PROGRAM PRG_PLC2
VAR
	EncoderValue AT %I* : UINT;
	Pos					: LREAL;
END_VAR

F_ConsumeTime(20);

Pos:= UINT_TO_LREAL(EncoderValue)*100;

END_PROGRAM

(* stored: Version 1.1.0.1, ProductVersion 3.1.4026.18
   POU PRG_PLC2: Id {cce961d7-e523-4b2f-ba28-fed189464f30}, SpecialFunc None *)
